KUKA KRL program: reinigung.src, reinigung.dat

--- reinigung.src ---
&ACCESS RVO1
&REL 7
&COMMENT WARTUNGSPOS ANFAHREN
&PARAM TEMPLATE = C:\KRC\ROBOTER\TEMPLATE\VG_APPLPROG
&PARAM EDITMASK = *
DEF Reinigung( )
;FOLD INI;%{PE}%V3.2.0,%MKUKATPBASIS,%CINIT,%VCOMMON,%P
;FOLD BAS INI;%{E}%V3.2.0,%MKUKATPBASIS,%CINIT,%VINIT,%P
GLOBAL INTERRUPT DECL 3 WHEN $STOPMESS==TRUE DO IR_STOPM ( )
INTERRUPT ON 3
BAS (#INITMOV,0 )
;ENDFOLD (BAS INI)
;FOLD GRIPPER INI;%{E}%V3.2.0,%MKUKATPGRIPPER,%CINIT,%VINIT,%P
USER_GRP(0,DUMMY,DUMMY,GDEFAULT)
;ENDFOLD (GRIPPER INI)
;FOLD SPOT INI;%{E}%V3.2.0,%MKUKATPSPOT,%CINIT,%VINIT,%P
USERSPOT(#INIT)
;ENDFOLD (SPOT INI)
;FOLD USER INI;%{E}%V3.2.0,%MKUKATPUSER,%CINIT,%VINIT,%P
;Make your modifications here
;ENDFOLD (USER INI)
;ENDFOLD (INI)
;FOLD ; Anlagenbezeichn:               Stations-Nr:;%{PE}%R 3.2.24,%MKUKATPBASIS,%CCOMMENT,%VNORMAL,%P 2:Anlagenbezeichn:               Stations-Nr:
;ENDFOLD
;FOLD ; Stand / Version:;%{PE}%R 3.2.22,%MKUKATPBASIS,%CCOMMENT,%VNORMAL,%P 2:Stand / Version:
;ENDFOLD
;FOLD ; Name Bearbeiter:;%{PE}%R 3.2.22,%MKUKATPBASIS,%CCOMMENT,%VNORMAL,%P 2:Name Bearbeiter:
;ENDFOLD
;Ueberpruefung ob richtiges Werkzeug angedockt
CHK_W1_Wechs_OK()
;FOLD PTP HOME  Vel= 100 % DEFAULT;%{PE}%V3.2.0,%MKUKATPBASIS,%CMOVE,%VPTP,%P 1:PTP, 2:HOME, 3:, 5:100, 7:DEFAULT
    $BWDSTART = FALSE
    $H_POS=XHOME
    PDAT_ACT=PDEFAULT
    BAS (#PTP_DAT )
    FDAT_ACT=FHOME
    BAS (#FRAMES )
    BAS (#VEL_PTP,100 )
    PTP  XHOME
;ENDFOLD
;FOLD OUT 818 'SonderPos. erreicht'  State= FALSE ;%{PE}%R 3.2.43,%MKUKATPBASIS,%COUT,%VOUTX,%P 2:818, 5:FALSE, 6:
$OUT[818]=FALSE
;ENDFOLD
;FOLD WAIT FOR IN 818 'Anford. SonderPos.'  State= TRUE ;%{PE}%R 3.2.43,%MKUKATPBASIS,%CWAIT_FOR,%VWAIT_FOR,%P 1:0, 2:818, 5:TRUE, 6:
WAIT FOR $IN[818]==TRUE
;ENDFOLD

;FOLD PTP P1 CONT Vel= 100 % PDAT Tool[1] Base[0];%{PE}%R 3.2.43,%MKUKATPBASIS,%CMOVE,%VPTP,%P 1:PTP, 2:P1, 3:C_PTP, 5:100, 7:PDAT
    $BWDSTART = FALSE
    PDAT_ACT=PPDAT
    BAS(#PTP_DAT)
    FDAT_ACT=FP1
    BAS(#FRAMES)
    BAS(#VEL_PTP,100)
    PTP XP1 C_PTP
;ENDFOLD
;FOLD PTP P2 CONT Vel= 100 % PDAT Tool[1] Base[0];%{PE}%R 3.2.43,%MKUKATPBASIS,%CMOVE,%VPTP,%P 1:PTP, 2:P2, 3:C_PTP, 5:100, 7:PDAT
    $BWDSTART = FALSE
    PDAT_ACT=PPDAT
    BAS(#PTP_DAT)
    FDAT_ACT=FP2
    BAS(#FRAMES)
    BAS(#VEL_PTP,100)
    PTP XP2 C_PTP
;ENDFOLD

;\\--- Reinigungspos ist abhaengig ob Rob-Werkzeug mit
;\\--- gereinigt oder freigefahren wird (geschuetzt)
;FOLD PTP ReinigungsPos  Vel= 100 % PDAT Tool[1] Base[0];%{PE}%R 3.2.43,%MKUKATPBASIS,%CMOVE,%VPTP,%P 1:PTP, 2:ReinigungsPos, 3:, 5:100, 7:PDAT
    $BWDSTART = FALSE
    PDAT_ACT=PPDAT
    BAS(#PTP_DAT)
    FDAT_ACT=FReinigungsPos
    BAS(#FRAMES)
    BAS(#VEL_PTP,100)
    PTP XReinigungsPos
;ENDFOLD

;FOLD OUT 818 'SonderPos. erreicht'  State= TRUE ;%{PE}%R 3.2.43,%MKUKATPBASIS,%COUT,%VOUTX,%P 2:818, 5:TRUE, 6:
$OUT[818]=TRUE
;ENDFOLD
;FOLD WAIT FOR IN 818 'Anford. SonderPos.'  State= FALSE ;%{PE}%R 3.2.43,%MKUKATPBASIS,%CWAIT_FOR,%VWAIT_FOR,%P 1:0, 2:818, 5:FALSE, 6:
WAIT FOR $IN[818]==FALSE
;ENDFOLD

;FOLD PTP P3 CONT Vel= 100 % PDAT Tool[1] Base[0];%{PE}%R 3.2.43,%MKUKATPBASIS,%CMOVE,%VPTP,%P 1:PTP, 2:P3, 3:C_PTP, 5:100, 7:PDAT
    $BWDSTART = FALSE
    PDAT_ACT=PPDAT
    BAS(#PTP_DAT)
    FDAT_ACT=FP3
    BAS(#FRAMES)
    BAS(#VEL_PTP,100)
    PTP XP3 C_PTP
;ENDFOLD
;FOLD PTP P4 CONT Vel= 100 % PDAT Tool[1] Base[0];%{PE}%R 3.2.43,%MKUKATPBASIS,%CMOVE,%VPTP,%P 1:PTP, 2:P4, 3:C_PTP, 5:100, 7:PDAT
    $BWDSTART = FALSE
    PDAT_ACT=PPDAT
    BAS(#PTP_DAT)
    FDAT_ACT=FP4
    BAS(#FRAMES)
    BAS(#VEL_PTP,100)
    PTP XP4 C_PTP
;ENDFOLD
;FOLD PTP HOME  Vel= 100 % DEFAULT;%{PE}%R 3.2.24,%MKUKATPBASIS,%CMOVE,%VPTP,%P 1:PTP, 2:HOME, 3:, 5:100, 7:DEFAULT
    $BWDSTART = FALSE
    PDAT_ACT=PDEFAULT
    BAS(#PTP_DAT)
    FDAT_ACT=FHOME
    BAS(#FRAMES)
    BAS(#VEL_PTP,100)
    $H_POS=XHOME
    PTP XHOME
;ENDFOLD

;FOLD OUT 818 'SonderPos. erreicht'  State= FALSE ;%{PE}%R 3.2.43,%MKUKATPBASIS,%COUT,%VOUTX,%P 2:818, 5:FALSE, 6:
$OUT[818]=FALSE
;ENDFOLD
;FOLD WAIT FOR IN 818 'Anford. SonderPos.'  State= FALSE ;%{PE}%R 3.2.43,%MKUKATPBASIS,%CWAIT_FOR,%VWAIT_FOR,%P 1:0, 2:818, 5:FALSE, 6:
WAIT FOR $IN[818]==FALSE
;ENDFOLD
END

--- reinigung.dat ---
&ACCESS RVO1
&REL 7
&COMMENT WARTUNGSPOS ANFAHREN
&PARAM TEMPLATE = C:\KRC\ROBOTER\TEMPLATE\VG_APPLPROG
&PARAM EDITMASK = *
DEFDAT  REINIGUNG
;FOLD EXTERNAL DECLARATIONS;%{PE}%V3.2.0,%MKUKATPBASIS,%CEXT,%VCOMMON,%P
;FOLD BAS EXT;%{PE}%V3.2.0,%MKUKATPBASIS,%CEXT,%VEXT,%P
EXT  BAS (BAS_COMMAND  :IN,REAL  :IN )
DECL INT SUCCESS
;ENDFOLD
;FOLD A10 EXT;%{E}%V3.2.0,%MKUKATPARC,%CEXT,%VEXT,%P
EXT  A10 (A_CMD_T:IN,A_STRT_T:IN,A_WELD_T:IN,A_END_T:IN,INT:IN)
;ENDFOLD
;FOLD A20 EXT;%{E}%V3.2.0,%MKUKATPA20,%CEXT,%VEXT,%P
EXT  A20 (INT  :IN,WELD_ST:IN,WELD_FI:IN,INT:IN)
;ENDFOLD
;FOLD GRIPPER EXT;%{E}%V3.2.0,%MKUKATPGRIPPER,%CEXT,%VEXT,%P
EXT  H50 (INT:IN, INT:IN ,INT:IN ,GRP_TYP:IN)
;ENDFOLD
;FOLD SPOT EXT;%{E}%V3.2.0,%MKUKATPSPOT,%CEXT,%VEXT,%P
EXT  USERSPOT (S_COMMAND  :IN, SPOT_TYPE:IN)
;ENDFOLD
;FOLD TOUCHSENSE EXT;%{E}%V3.2.0,%MKUKATPTS,%CEXT,%VEXT,%P
EXT  H70 (INT  :IN,SRCH_TYP_2  :OUT,E6POS  :IN,SRCH_TYP_3  :IN,SRCH_TYP_2  :IN,SRCH_TYP_2  :IN,SRCH_TYP_2  :IN,SRCH_TYP_2  :IN,SRCH_TYP_2  :IN,INT  :IN )
;ENDFOLD
;FOLD USER EXT;%{E}%V3.2.0,%MKUKATPUSER,%CEXT,%VEXT,%P
;Make here your modifications
;FOLD DC_BOLZEN_V3.01 ;%{}%V3.2.0,%MKUKATPUSER,%CEXT,%VEXT,%P
;EXT  BOLZEN (CALLMODE_T  :IN,INT  :IN,INT  :IN,INT  :IN,INT  :IN )
;ENDFOLD
;FOLD COLLISION_V3.01 ;%{}%V3.2.0,%MKUKATPUSER,%CEXT,%VEXT,%P
EXT  COLLSTOP (INT  :IN,INT  :IN )
;ENDFOLD
;ENDFOLD
;ENDFOLD

DECL BASIS_SUGG_T LAST_BASIS={POINT1[] "P0                      ",POINT2[] "P0                      ",CP_PARAMS[] "CPDAT0                  ",PTP_PARAMS[] "PDAT0                  ",CONT[] "                        ",CP_VEL[] "2                       ",PTP_VEL[] "100                     "}
DECL E6POS XP1={x 2620.467,y -20.40036,z 887.2352,a -77.88962,b 89.39492,c -77.42761,s 4,t 24,e1 0.0,e2 0.0,e3 0.0,e4 0.0,e5 0.0,e6 0.0}
DECL E6POS XP2={x 2620.467,y -20.40036,z 887.2352,a -77.88962,b 89.39492,c -77.42761,s 4,t 24,e1 0.0,e2 0.0,e3 0.0,e4 0.0,e5 0.0,e6 0.0}
DECL E6POS XWARTUNGSPOS={x 2620.467,y -20.40036,z 887.2352,a -77.88962,b 89.39492,c -77.42761,s 4,t 24,e1 0.0,e2 0.0,e3 0.0,e4 0.0,e5 0.0,e6 0.0}
DECL E6POS XP3={x 2620.467,y -20.40036,z 887.2352,a -77.88962,b 89.39492,c -77.42761,s 4,t 24,e1 0.0,e2 0.0,e3 0.0,e4 0.0,e5 0.0,e6 0.0}
DECL E6POS XP4={x 2620.467,y -20.40036,z 887.2352,a -77.88962,b 89.39492,c -77.42761,s 4,t 24,e1 0.0,e2 0.0,e3 0.0,e4 0.0,e5 0.0,e6 0.0}
DECL E6POS XReinigungsPos={x 2620.467,y -20.40036,z 887.2352,a -77.88962,b 89.39492,c -77.42761,s 4,t 24,e1 0.0,e2 0.0,e3 0.0,e4 0.0,e5 0.0,e6 0.0}
DECL FDAT FP1={TOOL_NO 1,BASE_NO 0,IPO_FRAME #BASE}
DECL PDAT PPDAT={VEL 100.0,ACC 100.0,APO_DIST 100.0}
DECL FDAT FP2={TOOL_NO 1,BASE_NO 0,IPO_FRAME #BASE}
DECL FDAT FWartungsPos={TOOL_NO 1,BASE_NO 0,IPO_FRAME #BASE}
DECL FDAT FP3={TOOL_NO 1,BASE_NO 0,IPO_FRAME #BASE}
DECL FDAT FP4={TOOL_NO 1,BASE_NO 0,IPO_FRAME #BASE}
DECL FDAT FReinigungsPos={TOOL_NO 1,BASE_NO 0,IPO_FRAME #BASE}
ENDDAT
